// TIA Portal V17 export
// export: Created 2022-06-27T13:56:49.8989339Z, ExportSetting WithDefaults, DisplayName Totally Integrated Automation Portal, DisplayVersion V17 Update 3, DisplayName TIA Portal Openness, DisplayVersion V17 Update 3, DisplayName TIA Portal Version Control Interface, DisplayVersion V17, DisplayName SINAMICS Startdrive Advanced, DisplayVersion V17 Update1, DisplayName SINAMICS Startdrive G110M, G120, G120C, G120D, G120P, G115D, DisplayVersion V17 Update1, DisplayName SINAMICS Startdrive G130, G150, S120, S150, SINAMICS MV, S210, DisplayVersion V17 Update1, DisplayName STEP 7 Professional, DisplayVersion V17 Update 3, DisplayName STEP 7 Safety, DisplayVersion V17, DisplayName WinCC UA Professional, DisplayVersion V17 Update 3
FUNCTION_BLOCK "S03_VALVES"   // FB3, LAD
{ S7_Optimized_Access := 'TRUE' }
VERSION : 0.1
// stored: AutoNumber false, IsIECCheckEnabled false, IsRetainMemResEnabled false, MemoryReserve 100, SetENOAutomatically false, UDAEnableTagReadback false
BEGIN

REGION Network 1: Calls all subfunctions
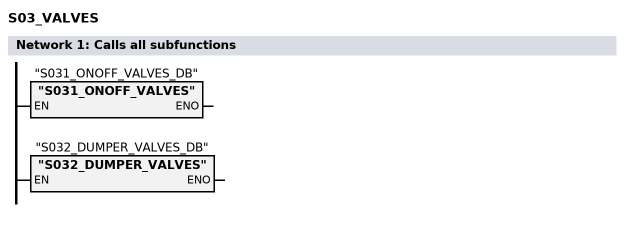
   RUNG wire#powerrail
      "S031_ONOFF_VALVES_DB"()
   END_RUNG
   RUNG wire#powerrail
      "S032_DUMPER_VALVES_DB"()
   END_RUNG
   // the same network as SCL:
   "S031_ONOFF_VALVES_DB"();   // "S031_ONOFF_VALVES"
   "S032_DUMPER_VALVES_DB"();   // "S032_DUMPER_VALVES"
END_REGION
END_FUNCTION_BLOCK
